// TIA Portal project "PrepaFormation" (V17)

(* hardware
DEVICE "S7-1200 station_1"  S7-1200 Station
   slot 0: "Rack_0"  S7-1200 Rack  Rack  V1.0
   slot 1: "PLC_1"  CPU 1211C DC/DC/Rly  6ES7 211-1HE40-0XB0  V4.5
   slot 3: "DQ 4x24VDC_1"  DQ4 signal board (200 kHz)  6ES7 222-1BD30-0XB0  V1.0
DEVICE "HMI_1"  KTP400 Comfort
   slot 0: "HMI_1"  KTP400 Comfort  6AV2 124-2DC01-0AX0  17.0.0.0
   slot 1: "HMI_RT_1"  KTP400 Comfort  6AV2 124-2DC01-0AX0  17.0.0.0
   slot 5: "HMI_1.IE_CP_1"  PROFINET Interface  17.0.0.0
      slot 1: "PROFINET Interface_1"  PROFINET Interface
         slot 1: "Port_1"  Port
   slot 7: "HMI_1.MPI/DP_CP_1"  MPI/DP Interface  17.0.0.0
DEVICE "ET 200SP SIPLUS_1"  ET 200SP-Station
   slot 0: "Rack_0"  Rack  6ES5 710-8MAx1
   slot 0: "IO device_1"  IM155-6 PN ST SIPLUS  6AG1 155-6AU00-7BN0  V3.3
      slot 1: "PROFINET interface"  6AG1 155-6AU00-7BN0
   slot 1: "DI 8x24VDC ST SIPLUS_1"  DI 8x24VDC ST SIPLUS  6AG1 131-6BF00-7BA0  V1.1
      slot 1: "DI 8x24VDC ST_1"  DI 8x24VDC ST
   slot 2: "DQ 4x24VDC/2A ST SIPLUS_1"  DQ 4x24VDC/2A ST SIPLUS  6AG1 132-6BD20-7BA0  V1.1
      slot 1: "DQ 4x24VDC/2A ST_1"  DQ 4x24VDC/2A ST
   slot 3: "AI 8xU BA SIPLUS_1"  AI 8xU BA SIPLUS  6AG1 134-6FF00-2AA1  V1.0
      slot 1: "AI 8xU BA_1"  AI 8xU BA
   slot 4: "AQ 2xI ST SIPLUS_1"  AQ 2xI ST SIPLUS  6AG1 135-6GB00-7BA1  V1.0
      slot 1: "AQ 2xI ST_1"  AQ 2xI ST
   slot 5: "CM PtP SIPLUS RAIL_1"  CM PtP SIPLUS RAIL  6AG2 137-6AA00-1BA0  V1.0
      slot 1: "CM PtP_1"  CM PtP Sub
   slot 6: "DS 0.1 - 0.4A HF 3DI/LC_1"  DS 0.1 - 0.4A HF 3DI/LC  3RK1 308-0AA00-0CP0  V1.2
      slot 1: "DS 0.1-0.4 A HF 3DI/LC_1"  DS 0.1-0.4 A HF 3DI/LC  3RK1 308-0AA00-0CP0 submodule
   slot 7: "Server module SIPLUS_1"  Server module SIPLUS  6AG1 193-6PA00-7AA0  V1.1
      slot 1: "Server module_1"  Server module
   slot 127: "BA 2xRJ45 SIPLUS"  BA 2xRJ45 SIPLUS  6AG1 193-6AR00-7AA0  V0.0
      slot 1: "Port_1"  X1 P1 R  6AG1 193-6AR00-7AA0  V0.0
      slot 2: "Port_2"  X1 P2 R  6AG1 193-6AR00-7AA0  V0.0
DEVICE "S7-1500/ET200MP station_1"  S7-1500 station
   slot 0: "Rail_0"  Rack  6ES7 590-1***0-0AA0
   slot 1: "PLC_2"  CPU 1511-1 PN  6ES7 511-1AK02-0AB0  V2.9
      slot 3: "CPU display_1"  6ES7591-1AA00-0AA0
      slot 32768: "PROFINET interface_1"  X1
         slot 32769: "Port_1"  X1 P1
         slot 32770: "Port_2"  X1 P2
      slot 34817: "Virtual CP interface port_1"  Virtual CP interface port  Virtual CP interface port
DEVICE "S7-1500/ET200MP station_2"  S7-1500 station
   slot 0: "Rail_0"  Rack  6ES7 590-1***0-0AA0
   slot 1: "PLC_3"  CPU 1515-2 PN  6ES7 515-2AM02-0AB0  V2.9
      slot 3: "CPU display_1"  6ES7591-1BA00-0AA0
      slot 32768: "PROFINET interface_1"  X1
         slot 32769: "Port_1"  X1 P1
         slot 32770: "Port_2"  X1 P2
      slot 33024: "PROFINET interface_2"  X2
         slot 33025: "Port_1"  X2 P1
      slot 34817: "Virtual CP interface port_1"  Virtual CP interface port  Virtual CP interface port
*)

// ===== PLC "PLC_1"  CPU 1211C DC/DC/Rly =====

VAR_GLOBAL   // PLC tag table "Default tag table"
   "Signal" AT %MW0 : UInt;
   "StartSignal" AT %M2.0 : Bool;
   "STartInc" AT %M2.1 : Bool;
   "StartDec" AT %M2.2 : Bool;
END_VAR

TYPE "Data_MBMaster"
   STRUCT
      busy : Bool;
      error : Bool;
      status : UDInt;
      data : Array[0..1] of Bool;
   END_STRUCT;
END_TYPE

DATA_BLOCK "Data"   // DB1
{ S7_Optimized_Access := 'FALSE' }
VERSION : 0.1
   VAR
      IHM_DATA : Struct
         Speed : Real;
         Position : Real;
         Acceleration : Real;
         Deceleration : Real;
      END_STRUCT;
      Data_Machine_ : Array[1..5] of Struct
         Speed : Real;
         Position : Real;
         Acceleration : Real;
         Deceleration : Real;
      END_STRUCT;
      Machine_No_From_HMI : UInt;
      Data_enter_Req_from_HMI : Bool;
   END_VAR
BEGIN
END_DATA_BLOCK

DATA_BLOCK "Data_Machine_handle_DB"   // DB2
{ S7_Optimized_Access := 'TRUE' }
VERSION : 0.1
// stored: InstanceOfName Data_Machine_handle
"Data_Machine_handle"
BEGIN
END_DATA_BLOCK

FUNCTION_BLOCK "Data_Machine_handle"   // FB1, LAD
{ S7_Optimized_Access := 'TRUE' }
VERSION : 0.1
   VAR_INPUT
      I_Machine_No : UInt;
      I_machine_Data_enter_Req : Bool;
   END_VAR
   VAR
      Old_Machine_No : UInt;
   END_VAR
BEGIN

REGION Network 1 (SCL)
   //IF #I_Machine_No <> #Old_Machine_No THEN
       // Statement section IF
       //"Data".IHM_DATA := "Data"."Data_Machine_"[#I_Machine_No];
       //#Old_Machine_No := #I_Machine_No;
   //END_IF;

   //IF #I_machine_Data_enter_Req THEN
       // Statement section IF
       //"Data"."Data_Machine_"[#I_Machine_No] := "Data".IHM_DATA;
   //END_IF;
END_REGION

REGION Network 2
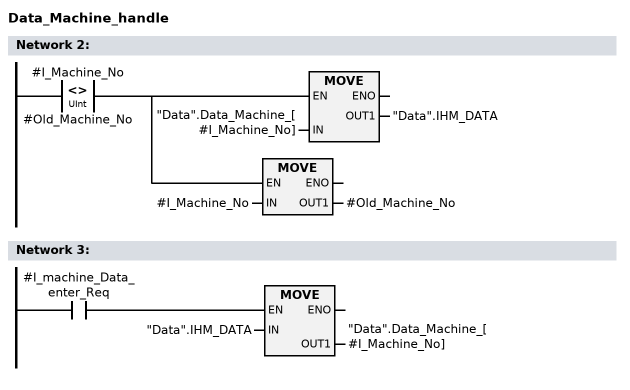
   RUNG wire#powerrail
      { S7_Templates := "SrcType := UInt" } NE_Contact(in1 := #I_Machine_No, in2 := #Old_Machine_No)
      wire#w1
      Move(in := "Data".Data_Machine_[#I_Machine_No], out1 => "Data".IHM_DATA)
   END_RUNG
   RUNG wire#w1
      Move(in := #I_Machine_No, out1 => #Old_Machine_No)
   END_RUNG
   // the same network as SCL:
   IF #I_Machine_No <> #Old_Machine_No THEN
       "Data".IHM_DATA := "Data".Data_Machine_[#I_Machine_No];
       #Old_Machine_No := #I_Machine_No;
   END_IF;
END_REGION

REGION Network 3
   RUNG wire#powerrail
      Contact( #I_machine_Data_enter_Req )
      Move(in := "Data".IHM_DATA, out1 => "Data".Data_Machine_[#I_Machine_No])
   END_RUNG
   // the same network as SCL:
   IF #I_machine_Data_enter_Req THEN "Data".Data_Machine_[#I_Machine_No] := "Data".IHM_DATA; END_IF;
END_REGION
END_FUNCTION_BLOCK

ORGANIZATION_BLOCK "Main"   // OB1, LAD, ProgramCycle
TITLE = "Main Program Sweep (Cycle)"
{ S7_Optimized_Access := 'TRUE' }
VERSION : 0.1
   VAR_INPUT
      Initial_Call : Bool;   // Initial call of this OB
      Remanence : Bool;   // =True, if remanent data are available
   END_VAR
BEGIN

REGION Network 1
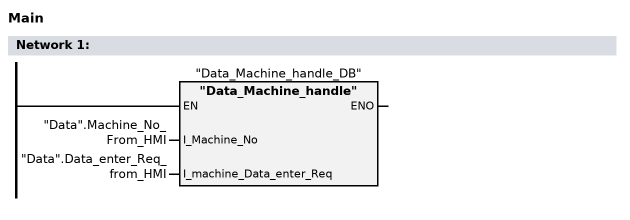
   RUNG wire#powerrail
      "Data_Machine_handle_DB"(I_Machine_No := "Data".Machine_No_From_HMI, I_machine_Data_enter_Req := "Data".Data_enter_Req_from_HMI)
   END_RUNG
   // the same network as SCL:
   "Data_Machine_handle_DB"(I_Machine_No := "Data".Machine_No_From_HMI,   // "Data_Machine_handle"
                           I_machine_Data_enter_Req := "Data".Data_enter_Req_from_HMI);
END_REGION
END_ORGANIZATION_BLOCK

ORGANIZATION_BLOCK "Block1s"   // OB30, LAD, CyclicInterrupt
{ S7_Optimized_Access := 'TRUE' }
VERSION : 0.1
   VAR_INPUT
      Initial_Call : Bool;   // Initial call of this OB
      Event_Count : Int;   // Events discarded
   END_VAR
BEGIN

REGION Network 1
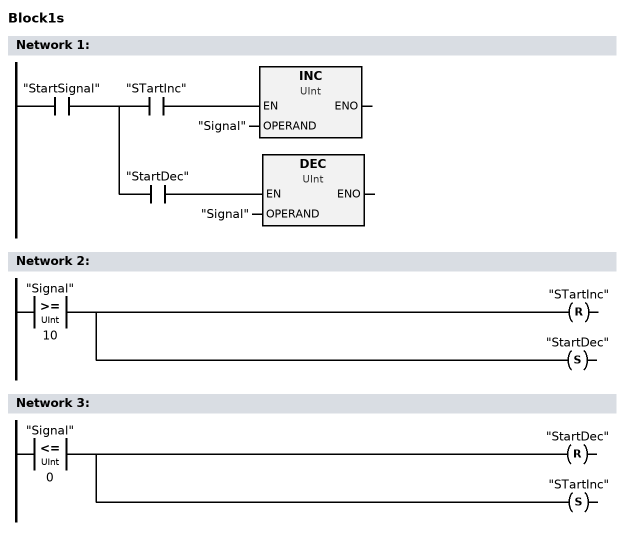
   RUNG wire#powerrail
      Contact( "StartSignal" )
      wire#w1
      Contact( "STartInc" )
      { S7_Templates := "DestType := UInt" } Inc( "Signal" )
   END_RUNG
   RUNG wire#w1
      Contact( "StartDec" )
      { S7_Templates := "DestType := UInt" } Dec( "Signal" )
   END_RUNG
   // the same network as SCL:
   IF "StartSignal" AND "STartInc" THEN "Signal" := "Signal" + 1; END_IF;
   IF "StartSignal" AND "StartDec" THEN "Signal" := "Signal" - 1; END_IF;
END_REGION

REGION Network 2
   RUNG wire#powerrail
      { S7_Templates := "SrcType := UInt" } GE_Contact(in1 := "Signal", in2 := 10)
      wire#w1
      R_Coil( "STartInc" )
   END_RUNG
   RUNG wire#w1
      S_Coil( "StartDec" )
   END_RUNG
   // the same network as SCL:
   IF "Signal" >= 10 THEN
       "STartInc" := FALSE;
       "StartDec" := TRUE;
   END_IF;
END_REGION

REGION Network 3
   RUNG wire#powerrail
      { S7_Templates := "SrcType := UInt" } LE_Contact(in1 := "Signal", in2 := 0)
      wire#w1
      R_Coil( "StartDec" )
   END_RUNG
   RUNG wire#w1
      S_Coil( "STartInc" )
   END_RUNG
   // the same network as SCL:
   IF "Signal" <= 0 THEN
       "StartDec" := FALSE;
       "STartInc" := TRUE;
   END_IF;
END_REGION
END_ORGANIZATION_BLOCK

ORGANIZATION_BLOCK "Startup"   // OB100, LAD, Startup
TITLE = "Complete Restart"
{ S7_Optimized_Access := 'TRUE' }
VERSION : 0.1
   VAR_INPUT
      LostRetentive : Bool;   // True if retentive data are lost
      LostRTC : Bool;   // True if date and time are lost
   END_VAR
BEGIN

REGION Network 1
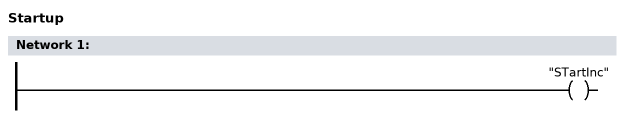
   RUNG wire#powerrail
      Coil( "STartInc" )
   END_RUNG
   // the same network as SCL:
   "STartInc" := TRUE;
END_REGION
END_ORGANIZATION_BLOCK

// ===== PLC "PLC_2"  CPU 1511-1 PN =====

ORGANIZATION_BLOCK "Main"   // OB1, LAD, ProgramCycle
TITLE = "Main Program Sweep (Cycle)"
{ S7_Optimized_Access := 'TRUE' }
VERSION : 0.1
   VAR_INPUT
      Initial_Call : Bool;   // Initial call of this OB
      Remanence : Bool;   // =True, if remanent data are available
   END_VAR
BEGIN
END_ORGANIZATION_BLOCK

// ===== PLC "PLC_3"  CPU 1515-2 PN =====

VAR_GLOBAL   // PLC tag table "Default tag table"
   "Tag_1" AT %I0.0 : Bool;
   "Tag_2" AT %M10.0 : Bool;
   "Tag_3" AT %M10.1 : Bool;
   "Tag_4" AT %M10.2 : Bool;
   "Tag_5" AT %M10.3 : Bool;
   "Tag_6" AT %M10.4 : Bool;
END_VAR

DATA_BLOCK "Block_1_DB"   // DB1
{ S7_Optimized_Access := 'TRUE' }
VERSION : 0.1
// stored: InstanceOfName Block_1
"Block_1"
BEGIN
END_DATA_BLOCK

FUNCTION_BLOCK "Block_1"   // FB1, GRAPH_PLUS
{ S7_Optimized_Access := 'TRUE' }
VERSION : 0.1
   VAR_INPUT
      OFF_SQ : Bool := false;   // Turn sequence off
      INIT_SQ : Bool := false;   // Set sequence to initial state
      ACK_EF : Bool := false;   // Acknowledge all errors and faults
      S_PREV : Bool := false;   // Output previous step in parameter S_NO
      S_NEXT : Bool := false;   // Indicate next step in parameter S_NO
      SW_AUTO : Bool := false;   // Automatic mode
      SW_TAP : Bool := false;   // Semiautomatic/switch with transition
      SW_TOP : Bool := false;   // Semiautomatic/ignore transition
      SW_MAN : Bool := false;   // Manual mode
      S_SEL : Int := 0;   // Select step to be output to S_NO
      S_ON : Bool := false;   // Activate step indicated in S_NO
      S_OFF : Bool := false;   // Deactivate step indicated S_NO
      T_PUSH : Bool := false;   // Enable transition to switch in semi automatic mode
   END_VAR
   VAR_OUTPUT
      S_NO : Int := 0;   // Step number
      S_MORE : Bool := false;   // More steps are available and can be shown in S_NO
      S_ACTIVE : Bool := false;   // Step indicated in S_NO is active
      ERR_FLT : Bool := false;   // Interlock or supervision group error
      AUTO_ON : Bool := false;   // Automatic mode is active
      TAP_ON : Bool := false;   // Semiautomatic mode/step with transition enabled
      TOP_ON : Bool := false;   // Semiautomatic mode/ignore transition enabled
      MAN_ON : Bool := false;   // Manual mode is active
   END_VAR
   VAR
      HMI_INFO : Array[0..8] of UInt;
      IF_PAR : G7_IfParPlus_V6;
      RT_DATA : G7_RTDataPlus_V6;   // Internal data area
      Trans1 : G7_TransitionPlus_V6;   // Transition structure
      Trans2 : G7_TransitionPlus_V6;   // Transition structure
      Trans3 : G7_TransitionPlus_V6;   // Transition structure
      Trans4 : G7_TransitionPlus_V6;   // Transition structure
      Trans5 : G7_TransitionPlus_V6;   // Transition structure
      Step1 : G7_StepPlus_V6;   // Step structure
      Step2 : G7_StepPlus_V6;   // Step structure
      Step3 : G7_StepPlus_V6;   // Step structure
      Step4 : G7_StepPlus_V6;   // Step structure
      Step5 : G7_StepPlus_V6;   // Step structure
      SINI : Array[0..1] of USInt;
      LSTT : Array[0..4] of USInt;
      ATAJ : Array[0..4] of USInt;
      ATAB : Array[0..4] of USInt;
      PSTT : Array[0..4] of USInt;
      NSTT : Array[0..4] of USInt;
      ASSJ : Array[0..4] of USInt;
      ASSB : Array[0..4] of USInt;
      PTTS : Array[0..4] of USInt;
      NTTS : Array[0..4] of USInt;
      SW_SQTS : Array[0..4] of USInt;
      SWITCH : Array[0..0] of USInt;
      TVX : Array[0..1] of USInt;
      TTX : Array[0..1] of USInt;
      TSX : Array[0..1] of USInt;
      S00X : Array[0..1] of USInt;
      SOFFX : Array[0..1] of USInt;
      SONX : Array[0..1] of USInt;
      SAX : Array[0..1] of USInt;
      SERRX : Array[0..5] of USInt;
      SMX : Array[0..5] of USInt;
      S0X : Array[0..5] of USInt;
      S1X : Array[0..5] of USInt;
      IL_ALARM_INST : Diag_Alarm;
      SUP_ALARM_INST : Diag_Alarm;
      STEP_TIME_ALARM_INST : Diag_Alarm;
      IEC_TIMER_INST : IEC_TIMER;
      TRANSACTION_FLAG : Bool := false;
   END_VAR
   // SINI[0] := 2;
   // LSTT[0] := 255;
   // LSTT[1] := 255;
   // LSTT[2] := 255;
   // LSTT[3] := 255;
   // ATAJ[1] := 1;
   // ATAJ[2] := 2;
   // ATAJ[3] := 3;
   // ATAJ[4] := 4;
   // ATAB[1] := 1;
   // ATAB[2] := 2;
   // ATAB[3] := 3;
   // ATAB[4] := 4;
   // PSTT[1] := 1;
   // PSTT[2] := 2;
   // PSTT[3] := 3;
   // PSTT[4] := 4;
   // NSTT[0] := 1;
   // NSTT[1] := 2;
   // NSTT[2] := 3;
   // NSTT[3] := 4;
   // ASSJ[1] := 1;
   // ASSJ[2] := 2;
   // ASSJ[3] := 3;
   // ASSJ[4] := 4;
   // ASSB[1] := 1;
   // ASSB[2] := 2;
   // ASSB[3] := 3;
   // ASSB[4] := 4;
   // PTTS[0] := 255;
   // PTTS[2] := 1;
   // PTTS[3] := 2;
   // PTTS[4] := 3;
   // NTTS[1] := 1;
   // NTTS[2] := 2;
   // NTTS[3] := 3;
   // NTTS[4] := 4;
   // TVX[0] := 16#1;
   // TTX[0] := 16#1;
   // TSX[0] := 16#1;
   // S00X[0] := 16#1;
   // SOFFX[0] := 16#1;
   // SONX[0] := 16#1;
   // SAX[0] := 16#1;
   // SERRX[0] := 16#1;
   // SMX[0] := 16#1;
   // S0X[0] := 16#1;
   // S1X[0] := 16#1;
BEGIN
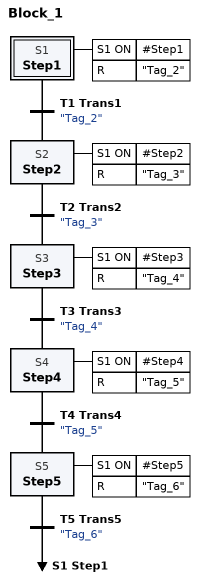
   // sequencer 1
   INITIAL_STEP Step1:   // S1, max time T#10S, warning time T#7S
          S1  ON   #Step1
              R    "Tag_2"
   END_STEP
   TRANSITION Trans1 FROM Step1 TO Step2   // T1
      := "Tag_2";
   END_TRANSITION
   STEP Step2:   // S2, max time T#10S, warning time T#7S
          S1  ON   #Step2
              R    "Tag_3"
   END_STEP
   TRANSITION Trans2 FROM Step2 TO Step3   // T2
      := "Tag_3";
   END_TRANSITION
   STEP Step3:   // S3, max time T#10S, warning time T#7S
          S1  ON   #Step3
              R    "Tag_4"
   END_STEP
   TRANSITION Trans3 FROM Step3 TO Step4   // T3
      := "Tag_4";
   END_TRANSITION
   STEP Step4:   // S4, max time T#10S, warning time T#7S
          S1  ON   #Step4
              R    "Tag_5"
   END_STEP
   TRANSITION Trans4 FROM Step4 TO Step5   // T4
      := "Tag_5";
   END_TRANSITION
   STEP Step5:   // S5, max time T#10S, warning time T#7S
          S1  ON   #Step5
              R    "Tag_6"
   END_STEP
   TRANSITION Trans5 FROM Step5 TO Step1   // T5, jump
      := "Tag_6";
   END_TRANSITION
END_FUNCTION_BLOCK

ORGANIZATION_BLOCK "Main"   // OB1, LAD, ProgramCycle
TITLE = "Main Program Sweep (Cycle)"
{ S7_Optimized_Access := 'TRUE' }
VERSION : 0.1
   VAR_INPUT
      Initial_Call : Bool;   // Initial call of this OB
      Remanence : Bool;   // =True, if remanent data are available
   END_VAR
BEGIN

REGION Network 1
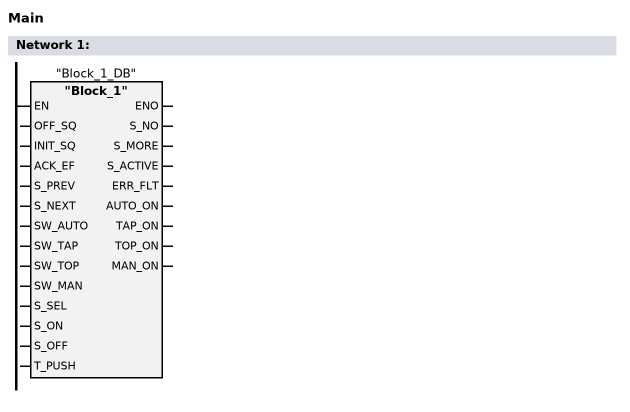
   RUNG wire#powerrail
      "Block_1_DB"(OFF_SQ :=, INIT_SQ :=, ACK_EF :=, S_PREV :=, S_NEXT :=, SW_AUTO :=, SW_TAP :=, SW_TOP :=, SW_MAN :=, S_SEL :=, S_ON :=, S_OFF :=, T_PUSH :=, S_NO =>, S_MORE =>, S_ACTIVE =>, ERR_FLT =>, AUTO_ON =>, TAP_ON =>, TOP_ON =>, MAN_ON =>)
   END_RUNG
   // the same network as SCL:
   "Block_1_DB"();   // "Block_1"
END_REGION
END_ORGANIZATION_BLOCK

(* ===== HMI "HMI_RT_1" =====
system functions are stored by id; their names below are inferred from use
connection "HMI_Connection_1": ETHERNET, S7_1200_OMS

HMI tags "Default tag table"
   "Data_IHM_DATA_Speed" : Real = PLC Data.IHM_DATA.Speed AT %DB1.DBD0, 1 s
   "Data_IHM_DATA_Position" : Real = PLC Data.IHM_DATA.Position AT %DB1.DBD4, 1 s
   "Data_IHM_DATA_Acceleration" : Real = PLC Data.IHM_DATA.Acceleration AT %DB1.DBD8, 1 s
   "Data_IHM_DATA_Deceleration" : Real = PLC Data.IHM_DATA.Deceleration AT %DB1.DBD12, 1 s
   "Data_Machine_No_From_HMI" : UInt = PLC Data.Machine_No_From_HMI AT %DB1.DBW96, 1 s
   "Data_Data_enter_Req_from_HMI" : Bool = PLC Data.Data_enter_Req_from_HMI AT %DB1.DBX98.0, 1 s

text list "Text_list_1": 0 'Select Machine No'; 1 'Machine No 1'; 2 'Machine No 2'; 3 'Machine No 3'; 4 'Machine No 4'; 5 'Machine No 5'

Template "Template_1" 480x272
   Button "Template_Button" at 415,70 size 63x63; TextOff 'Text'
   Button "Template_Button_1" at 415,138 size 63x63; TextOff 'Text'
   Button "Exit" at 415,207 size 63x63; TextOff 'Exit'; PictureOff "ExitRuntime_KTP400_Comfort_TR"; PictureOn "ExitRuntime_KTP400_Comfort_TR"
      on Release: StopRuntime(0)
   Button "Start screen" at 415,1 size 63x63; TextOff 'Start screen'; PictureOff "NavigateHome_KTP400_Comfort_TR"; PictureOn "NavigateHome_KTP400_Comfort_TR"
      on Release: ActivateScreen("Root screen", 0)

screen "Root screen" 480x272, template "Template_1"
   SymbolicIOField "Symbolic I/O field_1" at 14,14 size 183x32; TextOff '0'; TextOn '1'; TextList "Text_list_1"
      ProcessValue <- "Data_Machine_No_From_HMI"
   IOField "I/O field_1" at 18,65 size 96x32; FormatPattern 9999
      ProcessValue <- "Data_IHM_DATA_Speed"
   IOField "I/O field_2" at 18,114 size 96x32; FormatPattern 9999
      ProcessValue <- "Data_IHM_DATA_Position"
   IOField "I/O field_3" at 18,167 size 96x32; FormatPattern 9999
      ProcessValue <- "Data_IHM_DATA_Acceleration"
   IOField "I/O field_4" at 18,222 size 96x32; FormatPattern 9999
      ProcessValue <- "Data_IHM_DATA_Deceleration"
   TextField "Text field_1" at 137,67 size 85x20; Text 'Speed'
   TextField "Text field_2" at 131,123 size 109x20; Text 'Position'
   TextField "Text field_3" at 129,171 size 140x20; Text 'Acceleration'
   TextField "Text field_4" at 133,223 size 141x20; Text 'deceleration'
   Button "Button_1" at 223,19 size 139x32; TextOff 'Enter DATA'; Authorization "Operate"
      on Release: ResetBit("Data_Data_enter_Req_from_HMI")
      on Press: SetBit("Data_Data_enter_Req_from_HMI")

screen "Screen_1" 480x272
   Button "FB_2ArrowsDown_Rectangular" at 153,56 size 80x50; TextOff 'Text'; PictureOn "FB_2ArrowsDown_Rectangular_Pressed_256c"; PictureOff "FB_2ArrowsDown_Rectangular_Released_256c"
   Switch "Toggle_Horizontal_G" at 158,155 size 80x50; CaptionText 'Switch'; TextOff '0'; TextOn '1'; PictureOff "Toggle_Horizontal_G_Off_256c"; PictureOn "Toggle_Horizontal_G_On_256c"
   Switch "Pushbutton_Round_G" at 351,117 size 50x50; CaptionText 'Switch'; TextOff '0'; TextOn '1'; PictureOff "Pushbutton_Round_G_Off_256c"; PictureOn "Pushbutton_Round_G_On_256c"
   Switch "Pushbutton_Emergency" at 285,32 size 80x80; CaptionText 'Switch'; TextOff '0'; TextOn '1'; PictureOff "Pushbutton_Emergency_Off_256c"; PictureOn "Pushbutton_Emergency_On_256c"
   Switch "Lever_Vertical_1" at 351,186 size 50x80; CaptionText 'Switch'; TextOff '0'; TextOn '1'; PictureOff "Lever_Vertical_1_Off_256c"; PictureOn "Lever_Vertical_1_On_256c"
*)